PROGRAM MAIN
VAR
END_VAR

//This is a test
//

END_PROGRAM

(* stored: Version 1.1.0.1, ProductVersion 3.1.4024.12
   POU MAIN: Id {3e8521a1-8705-4303-9e18-c70ec2ab17f6}, SpecialFunc None *)
